FUNCTION Convert_ULINT_TO_TIME : Hresult
VAR_INPUT
	in : ULINT;
	out : REFERENCE TO TIME;
END_VAR
VAR
	converted : TIME;
END_VAR

converted := ULINT_TO_TIME(in);

IF (TIME_TO_ULINT(converted) <> in) THEN
	Convert_ULINT_TO_TIME := INCOMPATIBLE;
	RETURN;
END_IF

out := converted;

END_FUNCTION

(* stored: Version 1.1.0.1, ProductVersion 3.1.4024.12
   POU Convert_ULINT_TO_TIME: Id {6704fff0-c480-46d6-b9c4-11074b8fd8ec}, SpecialFunc None *)
